FUNCTION_BLOCK PlotterOverallStateMachine (* Template for a simple Basic Function Block Type *)
  (* Standard: 61499-2 *)
  (* Version 1.0, 2020-02-20, Mario *)
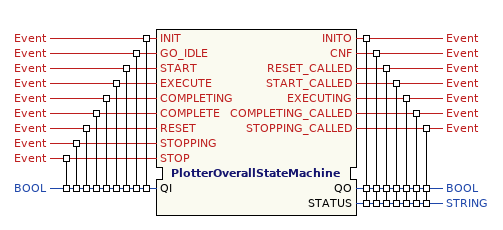
  EVENT_INPUT
    INIT WITH QI; (* Initialization Request *)
    GO_IDLE WITH QI;
    START WITH QI;
    EXECUTE WITH QI;
    COMPLETING WITH QI;
    COMPLETE WITH QI;
    RESET WITH QI;
    STOPPING WITH QI;
    STOP WITH QI;
  END_EVENT
  EVENT_OUTPUT
    INITO WITH QO, STATUS; (* Initialization Confirm *)
    CNF WITH QO, STATUS; (* Execution Confirmation *)
    RESET_CALLED WITH QO, STATUS;
    START_CALLED WITH QO, STATUS;
    EXECUTING WITH QO, STATUS;
    COMPLETING_CALLED WITH QO, STATUS;
    STOPPING_CALLED WITH QO, STATUS;
  END_EVENT
  VAR_INPUT
    QI : BOOL; (* Input event qualifier *)
  END_VAR
  VAR_OUTPUT
    QO : BOOL; (* Output event qualifier *)
    STATUS : STRING;
  END_VAR
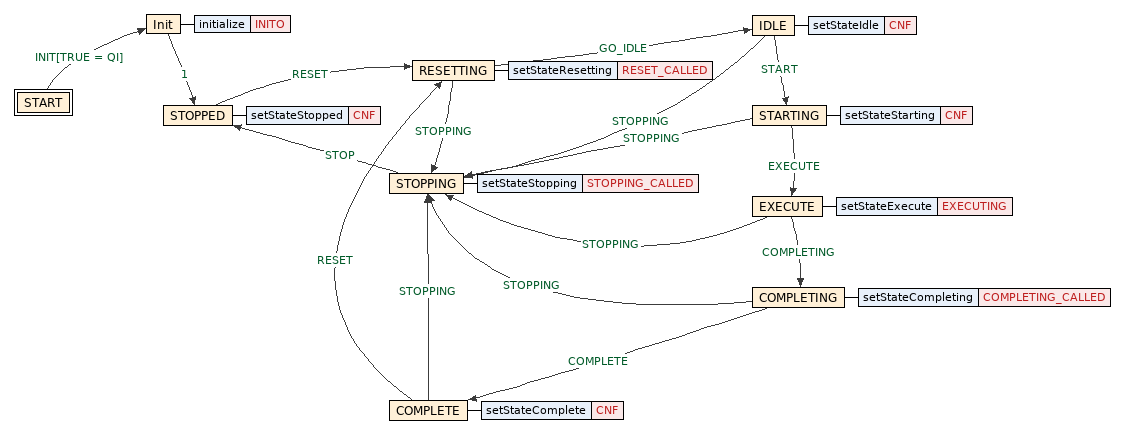
  EC_STATES
    START; (* Initial State *)
    Init : initialize -> INITO; (* Initialization *)
    RESETTING : setStateResetting -> RESET_CALLED;
    EXECUTE : setStateExecute -> EXECUTING;
    COMPLETING : setStateCompleting -> COMPLETING_CALLED;
    COMPLETE : setStateComplete -> CNF;
    STARTING : setStateStarting -> CNF;
    IDLE : setStateIdle -> CNF;
    STOPPING : setStateStopping -> STOPPING_CALLED;
    STOPPED : setStateStopped -> CNF;
  END_STATES
  EC_TRANSITIONS
    START TO Init := INIT[TRUE = QI];
    Init TO STOPPED := 1;
    IDLE TO STOPPING := STOPPING;
    STARTING TO STOPPING := STOPPING;
    EXECUTE TO STOPPING := STOPPING;
    COMPLETING TO STOPPING := STOPPING;
    COMPLETE TO STOPPING := STOPPING;
    RESETTING TO STOPPING := STOPPING;
    STOPPING TO STOPPED := STOP;
    STOPPED TO RESETTING := RESET;
    IDLE TO STARTING := START;
    STARTING TO EXECUTE := EXECUTE;
    COMPLETE TO RESETTING := RESET;
    RESETTING TO IDLE := GO_IDLE;
    EXECUTE TO COMPLETING := COMPLETING;
    COMPLETING TO COMPLETE := COMPLETE;
  END_TRANSITIONS
  ALGORITHM initialize IN ST: (* Initialization algorithm *)
QO := QI;
  END_ALGORITHM
  ALGORITHM deInitialize IN ST: (* Normally executed algorithm *)
QO := FALSE;
  END_ALGORITHM
  ALGORITHM normalOperation IN ST: (* new algorithm *)
QO := QI;

IF TRUE  = QI THEN
  (*  only perform normal operation of QI is true*)

END_IF;
  END_ALGORITHM
  ALGORITHM setStateIdle IN ST: (* new algorithm *)
STATUS := "IDLE";
  END_ALGORITHM
  ALGORITHM setStateStarting IN ST: (* new algorithm *)
STATUS := "STARTING";
  END_ALGORITHM
  ALGORITHM setStateExecute IN ST: (* new algorithm *)
STATUS := "EXECUTE";
  END_ALGORITHM
  ALGORITHM setStateCompleting IN ST: (* new algorithm *)
STATUS := "COMPLETING";
  END_ALGORITHM
  ALGORITHM setStateComplete IN ST: (* new algorithm *)
STATUS := "COMPLETE";
  END_ALGORITHM
  ALGORITHM setStateResetting IN ST: (* new algorithm *)
STATUS := "RESETTING";
  END_ALGORITHM
  ALGORITHM setStateStopping IN ST: (* new algorithm *)
STATUS := "STOPPING";
  END_ALGORITHM
  ALGORITHM setStateStopped IN ST: (* new algorithm *)
STATUS := "STOPPED";
  END_ALGORITHM
END_FUNCTION_BLOCK
